///Checks if the HRESULT is error
FUNCTION Fail : BOOL
VAR_INPUT
    hr : HRESULT;
END_VAR
VAR
END_VAR

Fail := (hr < 0);

END_FUNCTION

(* stored: Version 1.1.0.1, ProductVersion 3.1.4020.12
   POU Fail: Id {8ce76036-fc0e-4632-93a1-4d7fa7219091}, SpecialFunc None *)
